TYPE E_Color :
(
    NONE := 0,
    RED := 1,
    BLUE := 2,
	YELLOW := 3,
    UNKNOWN := 4
);
END_TYPE

(* stored: Version 1.1.0.1
   DUT E_Color: Id {acac7edc-b9c3-4c5e-9035-440495015032} *)
